// TIA Portal V18 export
FUNCTION_BLOCK "FB10-Condition Check"   // FB10, LAD
{ S7_Optimized_Access := 'TRUE' }
VERSION : 0.1
// stored: AutoNumber false, IsIECCheckEnabled false, IsRetainMemResEnabled false, MemoryReserve 100, SetENOAutomatically false, UDAEnableTagReadback false
   VAR_INPUT
      "Time" : DInt;
      "Pump ON delay" : DInt;
      Check_Time { ExternalAccessible := 'False'; ExternalVisible := 'False'; ExternalWritable := 'False'} : DInt;
      Pressure_SP { ExternalAccessible := 'False'; ExternalVisible := 'False'; ExternalWritable := 'False'} : Real;
      Pressure_tolerance { ExternalAccessible := 'False'; ExternalVisible := 'False'; ExternalWritable := 'False'} : Real;
      Current_pressure { ExternalAccessible := 'False'; ExternalVisible := 'False'; ExternalWritable := 'False'} : Real;
      selected { ExternalAccessible := 'False'; ExternalVisible := 'False'; ExternalWritable := 'False'} : Bool;
   END_VAR
   VAR_OUTPUT
      "dispensing Time PV" : Int;
      "Checking Time pv" { ExternalAccessible := 'False'; ExternalVisible := 'False'; ExternalWritable := 'False'} : Int;
      test_ok { ExternalAccessible := 'False'; ExternalVisible := 'False'; ExternalWritable := 'False'} : Bool;
      test_nok { ExternalAccessible := 'False'; ExternalVisible := 'False'; ExternalWritable := 'False'} : Bool;
      test_fail { ExternalAccessible := 'False'; ExternalVisible := 'False'; ExternalWritable := 'False'} : Bool;
   END_VAR
   VAR_IN_OUT
      "Start ConditonCheck" : Bool;
      "Stop ConditonCheck" : Bool;
      "ConditonCheck Running" : Bool;
      "ConditonCheck completed" : Bool;
      "ON Gear Pump" : Bool;
      "ON inlet" : Bool;
   END_VAR
   VAR
      "dispensing time done" : Bool;
      "dispensing time in sec" : DInt;
      "timer in sec" : DInt;
      "timer PV in sec" : DInt;
      "timer input" : DInt;
      IEC_Timer_0_Instance { S7_SetPoint := 'True'} : TON_TIME;
      IEC_Timer_0_Instance_1 { S7_SetPoint := 'True'} : TON_TIME;
      IEC_Timer_0_Instance_2 { S7_SetPoint := 'True'} : TON_TIME;
      IEC_Timer_0_Instance_4 { S7_SetPoint := 'True'} : TON_TIME;
      "Press+ve" { ExternalAccessible := 'False'; ExternalVisible := 'False'; ExternalWritable := 'False'; S7_SetPoint := 'True'} : Real;
      "Press-ve" { ExternalAccessible := 'False'; ExternalVisible := 'False'; ExternalWritable := 'False'} : Real;
      IEC_Timer_0_Instance_3 { ExternalAccessible := 'False'; ExternalVisible := 'False'; ExternalWritable := 'False'; S7_SetPoint := 'True'} : TON_TIME;
      Checktime_ms { ExternalAccessible := 'False'; ExternalVisible := 'False'; ExternalWritable := 'False'; S7_SetPoint := 'True'} : DInt;
      Check_timesec { ExternalAccessible := 'False'; ExternalVisible := 'False'; ExternalWritable := 'False'} : DInt;
      temp_ons { ExternalAccessible := 'False'; ExternalVisible := 'False'; ExternalWritable := 'False'} : Bool;
   END_VAR
   VAR_TEMP   // added for the SCL form of the ladder/FBD networks
      _w1 : Bool;
   END_VAR
BEGIN

REGION Network 1
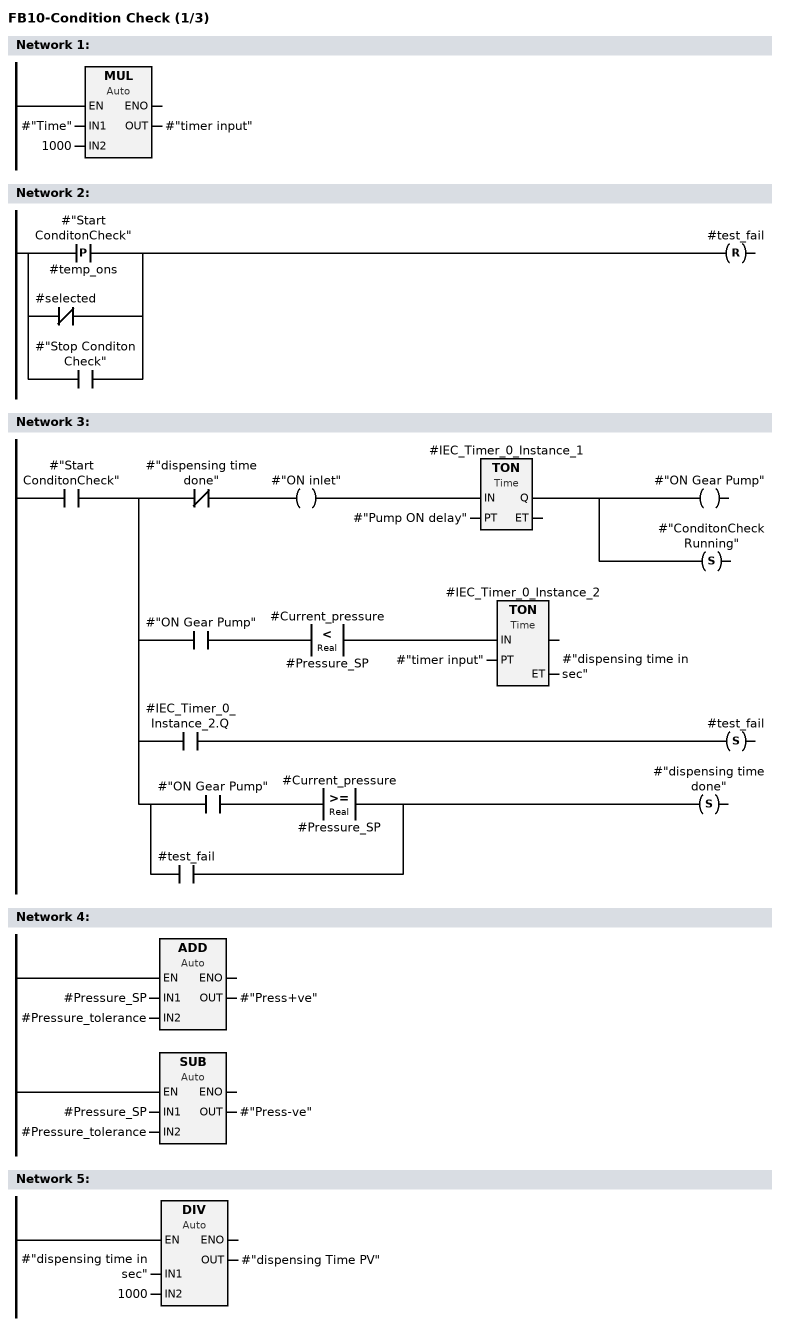
   RUNG wire#powerrail
      Mul(in1 := #"Time", in2 := 1000, out => #"timer input")
   END_RUNG
   // the same network as SCL:
   #"timer input" := #"Time" * 1000;
END_REGION

REGION Network 2
   RUNG wire#powerrail
      P_Contact(operand := #"Start ConditonCheck", bit := #temp_ons)
      wire#w1
      R_Coil( #test_fail )
   END_RUNG
   RUNG wire#powerrail
      I_Contact( #selected )
   END_RUNG wire#w1
   RUNG wire#powerrail
      Contact( #"Stop ConditonCheck" )
   END_RUNG wire#w1
   // the same network as SCL:
   #_w1 := #"Start ConditonCheck" AND NOT #temp_ons;   // rising edge of #"Start ConditonCheck"
   #temp_ons := #"Start ConditonCheck";
   IF #_w1 OR NOT #selected OR #"Stop ConditonCheck" THEN #test_fail := FALSE; END_IF;
END_REGION

REGION Network 3
   RUNG wire#powerrail
      Contact( #"Start ConditonCheck" )
      wire#w1
      I_Contact( #"dispensing time done" )
      Coil( #"ON inlet" )
      { S7_Templates := "time_type := Time" } #IEC_Timer_0_Instance_1.TON(pt := #"Pump ON delay", et =>)
      wire#w2
      Coil( #"ON Gear Pump" )
   END_RUNG
   RUNG wire#w2
      S_Coil( #"ConditonCheck Running" )
   END_RUNG
   RUNG wire#w1
      Contact( #"ON Gear Pump" )
      { S7_Templates := "SrcType := Real" } LT_Contact(in1 := #Current_pressure, in2 := #Pressure_SP)
      { S7_Templates := "time_type := Time" } #IEC_Timer_0_Instance_2.TON(pt := #"timer input", et => #"dispensing time in sec")
   END_RUNG
   RUNG wire#w1
      Contact( #IEC_Timer_0_Instance_2.Q )
      S_Coil( #test_fail )
   END_RUNG
   RUNG wire#w1
      Contact( #"ON Gear Pump" )
      { S7_Templates := "SrcType := Real" } GE_Contact(in1 := #Current_pressure, in2 := #Pressure_SP)
      wire#w3
      S_Coil( #"dispensing time done" )
   END_RUNG
   RUNG wire#w1
      Contact( #test_fail )
   END_RUNG wire#w3
   // the same network as SCL:
   #"ON inlet" := #"Start ConditonCheck" AND NOT #"dispensing time done";
   #IEC_Timer_0_Instance_1(IN := #"ON inlet", PT := #"Pump ON delay");   // TON
   #"ON Gear Pump" := #IEC_Timer_0_Instance_1.Q;
   IF #IEC_Timer_0_Instance_1.Q THEN #"ConditonCheck Running" := TRUE; END_IF;
   #IEC_Timer_0_Instance_2(IN := #"Start ConditonCheck" AND #"ON Gear Pump" AND (#Current_pressure < #Pressure_SP),   // TON
                           PT := #"timer input",
                           ET => #"dispensing time in sec");
   IF #"Start ConditonCheck" AND #IEC_Timer_0_Instance_2.Q THEN #test_fail := TRUE; END_IF;
   IF #"Start ConditonCheck" AND ((#"ON Gear Pump" AND (#Current_pressure >= #Pressure_SP)) OR #test_fail) THEN
       #"dispensing time done" := TRUE;
   END_IF;
END_REGION

REGION Network 4
   RUNG wire#powerrail
      Add(in1 := #Pressure_SP, in2 := #Pressure_tolerance, out => #"Press+ve")
   END_RUNG
   RUNG wire#powerrail
      Sub(in1 := #Pressure_SP, in2 := #Pressure_tolerance, out => #"Press-ve")
   END_RUNG
   // the same network as SCL:
   #"Press+ve" := #Pressure_SP + #Pressure_tolerance;
   #"Press-ve" := #Pressure_SP - #Pressure_tolerance;
END_REGION

REGION Network 5
   RUNG wire#powerrail
      Div(in1 := #"dispensing time in sec", in2 := 1000, out => #"dispensing Time PV")
   END_RUNG
   // the same network as SCL:
   #"dispensing Time PV" := #"dispensing time in sec" / 1000;
END_REGION

REGION Network 6
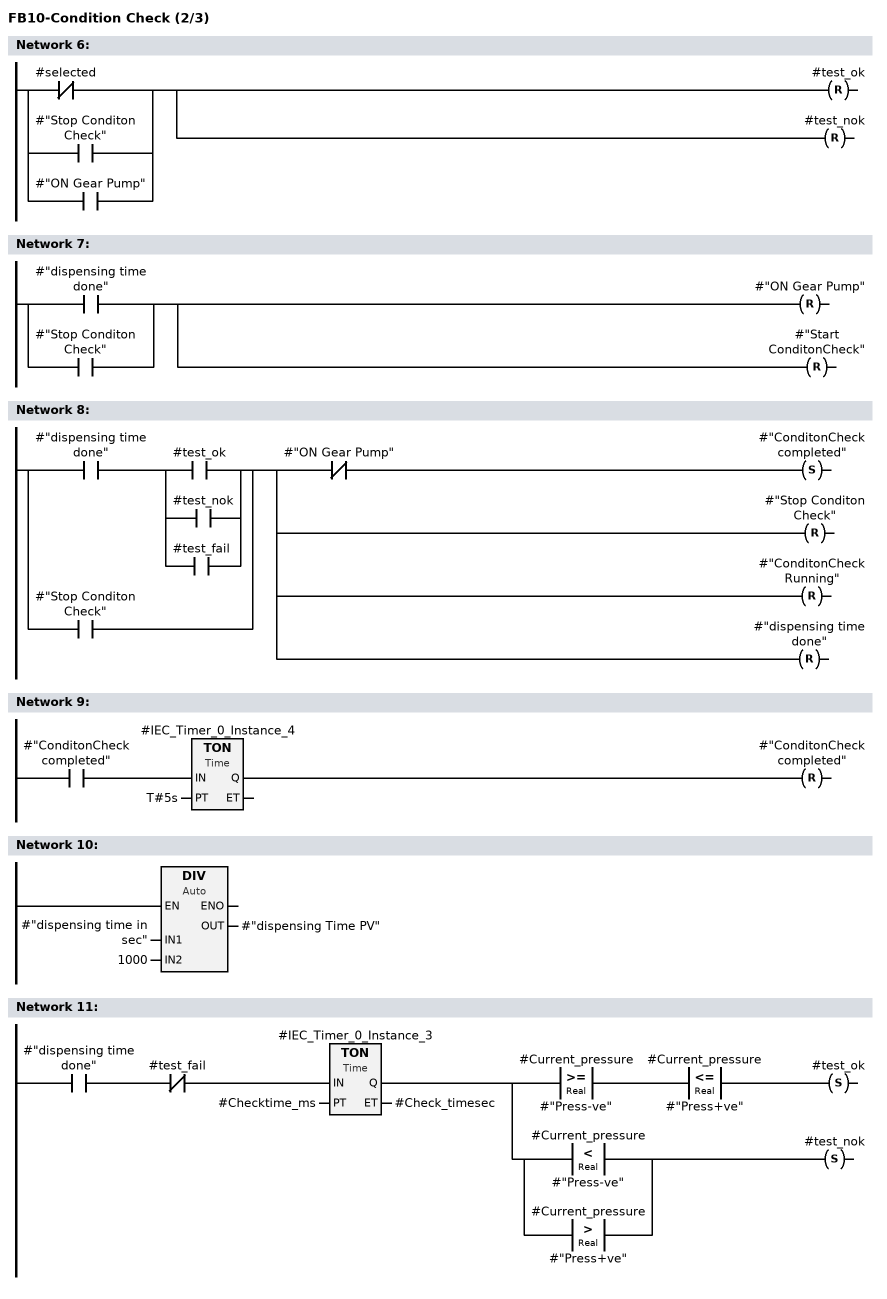
   RUNG wire#powerrail
      I_Contact( #selected )
      wire#w1
      R_Coil( #test_ok )
   END_RUNG
   RUNG wire#powerrail
      Contact( #"Stop ConditonCheck" )
   END_RUNG wire#w1
   RUNG wire#powerrail
      Contact( #"ON Gear Pump" )
   END_RUNG wire#w1
   RUNG wire#w1
      R_Coil( #test_nok )
   END_RUNG
   // the same network as SCL:
   IF NOT #selected OR #"Stop ConditonCheck" OR #"ON Gear Pump" THEN
       #test_ok := FALSE;
       #test_nok := FALSE;
   END_IF;
END_REGION

REGION Network 7
   RUNG wire#powerrail
      Contact( #"dispensing time done" )
      wire#w1
      R_Coil( #"ON Gear Pump" )
   END_RUNG
   RUNG wire#powerrail
      Contact( #"Stop ConditonCheck" )
   END_RUNG wire#w1
   RUNG wire#w1
      R_Coil( #"Start ConditonCheck" )
   END_RUNG
   // the same network as SCL:
   IF #"dispensing time done" OR #"Stop ConditonCheck" THEN
       #"ON Gear Pump" := FALSE;
       #"Start ConditonCheck" := FALSE;
   END_IF;
END_REGION

REGION Network 8
   RUNG wire#powerrail
      Contact( #"dispensing time done" )
      wire#w1
      Contact( #test_ok )
      wire#w2
      I_Contact( #"ON Gear Pump" )
      S_Coil( #"ConditonCheck completed" )
   END_RUNG
   RUNG wire#w1
      Contact( #test_nok )
   END_RUNG wire#w2
   RUNG wire#w1
      Contact( #test_fail )
   END_RUNG wire#w2
   RUNG wire#powerrail
      Contact( #"Stop ConditonCheck" )
   END_RUNG wire#w2
   RUNG wire#w2
      R_Coil( #"Stop ConditonCheck" )
   END_RUNG
   RUNG wire#w2
      R_Coil( #"ConditonCheck Running" )
   END_RUNG
   RUNG wire#w2
      R_Coil( #"dispensing time done" )
   END_RUNG
   // the same network as SCL:
   #_w1 := (#"dispensing time done" AND (#test_ok OR #test_nok OR #test_fail)) OR #"Stop ConditonCheck";
   IF #_w1 AND NOT #"ON Gear Pump" THEN #"ConditonCheck completed" := TRUE; END_IF;
   IF #_w1 THEN
       #"Stop ConditonCheck" := FALSE;
       #"ConditonCheck Running" := FALSE;
       #"dispensing time done" := FALSE;
   END_IF;
END_REGION

REGION Network 9
   RUNG wire#powerrail
      Contact( #"ConditonCheck completed" )
      { S7_Templates := "time_type := Time" } #IEC_Timer_0_Instance_4.TON(pt := T#5s, et =>)
      R_Coil( #"ConditonCheck completed" )
   END_RUNG
   // the same network as SCL:
   #IEC_Timer_0_Instance_4(IN := #"ConditonCheck completed", PT := T#5s);   // TON
   IF #IEC_Timer_0_Instance_4.Q THEN #"ConditonCheck completed" := FALSE; END_IF;
END_REGION

REGION Network 10
   RUNG wire#powerrail
      Div(in1 := #"dispensing time in sec", in2 := 1000, out => #"dispensing Time PV")
   END_RUNG
   // the same network as SCL:
   #"dispensing Time PV" := #"dispensing time in sec" / 1000;
END_REGION

REGION Network 11
   RUNG wire#powerrail
      Contact( #"dispensing time done" )
      I_Contact( #test_fail )
      { S7_Templates := "time_type := Time" } #IEC_Timer_0_Instance_3.TON(pt := #Checktime_ms, et => #Check_timesec)
      wire#w1
      { S7_Templates := "SrcType := Real" } GE_Contact(in1 := #Current_pressure, in2 := #"Press-ve")
      { S7_Templates := "SrcType := Real" } LE_Contact(in1 := #Current_pressure, in2 := #"Press+ve")
      S_Coil( #test_ok )
   END_RUNG
   RUNG wire#w1
      { S7_Templates := "SrcType := Real" } LT_Contact(in1 := #Current_pressure, in2 := #"Press-ve")
      wire#w2
      S_Coil( #test_nok )
   END_RUNG
   RUNG wire#w1
      { S7_Templates := "SrcType := Real" } GT_Contact(in1 := #Current_pressure, in2 := #"Press+ve")
   END_RUNG wire#w2
   // the same network as SCL:
   #IEC_Timer_0_Instance_3(IN := #"dispensing time done" AND NOT #test_fail,   // TON
                           PT := #Checktime_ms,
                           ET => #Check_timesec);
   IF #IEC_Timer_0_Instance_3.Q AND (#Current_pressure >= #"Press-ve") AND (#Current_pressure <= #"Press+ve") THEN
       #test_ok := TRUE;
   END_IF;
   IF #IEC_Timer_0_Instance_3.Q AND ((#Current_pressure < #"Press-ve") OR (#Current_pressure > #"Press+ve")) THEN
       #test_nok := TRUE;
   END_IF;
END_REGION

REGION Network 12
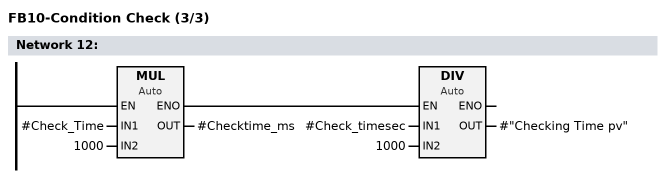
   RUNG wire#powerrail
      Mul(in1 := #Check_Time, in2 := 1000, out => #Checktime_ms)
      Div(in1 := #Check_timesec, in2 := 1000, out => #"Checking Time pv")
   END_RUNG
   // the same network as SCL:
   #Checktime_ms := #Check_Time * 1000;
   #"Checking Time pv" := #Check_timesec / 1000;
END_REGION
END_FUNCTION_BLOCK
